(* IEC 61131-3 sources: eCockpitGit/test_project/src/%F%00 Library/%F%Common Functions/%F%Linearsation/%F%ANY, 1 file *)

(* ---- %POU%FU_Linear2Ends.st ---- *)
//This is not finished
//This function, converts an x, value to an y value using and 2 points on the x and y scale
//This function has ends, which means the output is never greater or smaller than the range of y
// +-----------+----------+----------+-----------------------------------------------------------------------------------------------------------------------+
// |**Version**|**Author**| **Date** |**Changes**                                                                                                            |
// +-----------+----------+----------+-----------------------------------------------------------------------------------------------------------------------+
// | 1         | NSN      | 07-12-18 | Creation                                                                                                              |
// +-----------+----------+----------+-----------------------------------------------------------------------------------------------------------------------+
FUNCTION FU_Linear2Ends
VAR_INPUT
	XIn		:ANY;
	X1		:ANY;
	X2		:ANY;
	YOut	:ANY;
	Y1		:ANY;
	Y2		:ANY;
	Ends	:BOOL;
END_VAR
VAR
	a		:REAL;
	b		:REAL;
END_VAR
(*%!%__DELIMITER__%!%*)
